Universal Robots PolyScope program: force_simple_135.urp

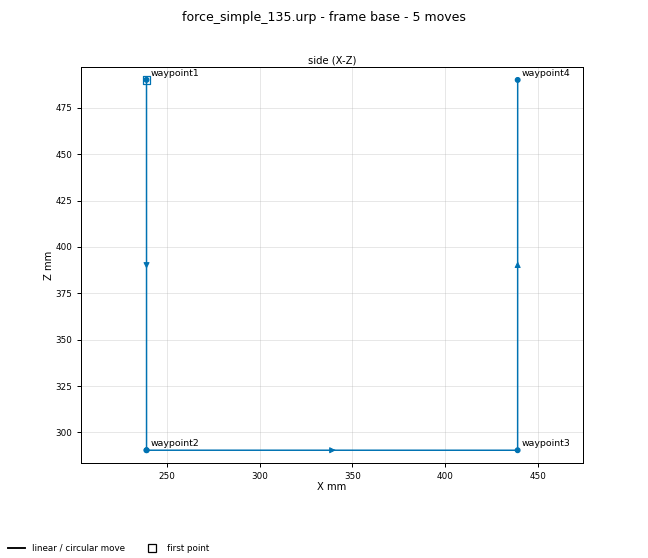
[picture p0: tool path of force_simple_135.urp in frame base, 5 of 5 moves have a stored position in this frame; points joined in program order, loops and branches not executed]
Program force_simple_135 (createdIn=3.2.19293 lastSavedIn=3.2.19293 directory=/programs installation=default robotSerialNumber=2015351391)
Calibrated DH parameters: a=[0.000352, -0.161198, -0.373486, 0.00005, 0.000049, 0]; d=[0.089268, 352.477598, -320.08558, -32.281492, 0.094939, 0.082518]; alpha=[1.570728, 0.001116, -0.003686, 1.571189, -1.570572, 0]; deltaTheta=[-0.000012, 1.181849, -1.491165, 0.309495, -0.000007, 0.000025]
Robot Program (runOnlyOnce=false motionType=MoveJ speed=1.047198 acceleration=1.396263 recalculateMotions=false)
  MoveL speed 250 mm/s, acceleration 1200 mm/s^2 (recalculateMotions=false) feature=Base
    Waypoint waypoint1: TCP in base x=239.017 y=198.815 z=490.017 mm, rx=0 ry=-3.1413 rz=-0.0001 rad; joints [60.677, -64.369, -100.788, -104.874, 89.744, 150.69] deg
    Waypoint waypoint2: TCP in base x=239.033 y=198.814 z=290.437 mm, rx=-0.0002 ry=-3.1413 rz=0 rad; joints [60.668, -64.345, -130.295, -75.396, 89.775, 150.583] deg
    Force Simple feature=Base; selection=[0, 0, 1, 0, 0, 0]; wrench=[0, 0, -30, 0, 0, 0]; limitsForce=[0.15, 0.15, 0.15, 1.047198, 1.047198, 1.047198]; limitsMotion=[0.1, 0.1, 0.1, 0.349066, 0.349066, 0.349066]
      Waypoint waypoint2: motionParameters(jointSpeed=1.047198 jointAcceleration=1.396263 cartesianSpeed=0.1 cartesianAcceleration=1.2); TCP in base x=239.033 y=198.814 z=290.437 mm, rx=-0.0002 ry=-3.1413 rz=0 rad; joints [60.668, -64.345, -130.295, -75.396, 89.775, 150.583] deg; flange x=239.018 y=198.806 z=490 mm, rx=-1.5849 ry=-0.1112 rz=-0.2808 rad
      Waypoint waypoint3: motionParameters(jointSpeed=1.047198 jointAcceleration=1.396263 cartesianSpeed=0.1 cartesianAcceleration=1.2); TCP in base x=439.004 y=198.816 z=290.42 mm, rx=-0.0001 ry=-3.1412 rz=0.0002 rad; joints [37.708, -91.084, -109.986, -68.975, 89.788, 127.574] deg
    Waypoint waypoint4: TCP in base x=439.028 y=198.806 z=489.974 mm, rx=0 ry=-3.1412 rz=0.0002 rad; joints [37.709, -88.125, -83.241, -98.68, 89.743, 127.675] deg
